# EPICS alarm handler configuration: apps/alhConfig/vacuum.alhConfig
GROUP    NULL                         VACUUM
CHANNEL  VACUUM                       hallb_VCG2C21Tr
$COMMAND  medm -x -attach -cmap -macro "sig=hallb_VCG2C21Tr" aiaocalc_alarm.adl >> /dev/null
$ALARMCOUNTFILTER  99 60
$GUIDANCE
                The cold cathode gauge at the moller region is out of spec.
                This means the vacuum between the shield wall and the tagger
                magnet has degraded.  Use the MYA Viewer and monitor the hallb_VCG2C21Tr
                to check for trends in the past few hours.  If the vacuum is degrading (values increasing on
                the plots) then contact engineering on call.   Also contact MCC and inform them about the
                problem, they might want to shut off the beam and close some valves to isolate the problem.
                If the vacuum spiked and recovered, continue taking
                data.
$END
CHANNEL  VACUUM                       hallb_VCG2C21ATr
$COMMAND  medm -x -attach -cmap -macro "sig=hallb_VCG2C21ATr" aiaocalc_alarm.adl >> /dev/null
$ALARMCOUNTFILTER  99 60
$GUIDANCE
                The cold cathode gauge at the moller region is out of spec.
                This means the vacuum between the shield wall and the tagger
                magnet has degraded.  Use the MYA Viewer and monitor the hallb_VCG2C21ATr
                to check for trends in the past few hours.  If the vacuum is degrading (values increasing on
                the plots) then contact engineering on call.   Also contact MCC and inform them about the
                problem, they might want to shut off the beam and close some valves to isolate the problem.
                If the vacuum spiked and recovered, continue taking
                data.
$END
CHANNEL  VACUUM                       hallb_VCG2C24ATr
$COMMAND  medm -x -attach -cmap -macro "sig=hallb_VCG2C24ATr" aiaocalc_alarm.adl >> /dev/null
$ALARMCOUNTFILTER  99 60
$GUIDANCE
                The tagger turbo speed is below operating range...it may have tripped off.
                Use the MYA Viewer and monitor hallb_VCG2C24ATr
                to check for trends in the past few hours.  If the vacuum is degrading (values increasing on
                the plots) then contact engineering on call.   Also contact MCC and inform them about the
                problem, they might want to shut off the beam and close some valves to isolate the problem.
                If the vacuum spiked and recovered, continue taking
                data.
$END
CHANNEL  VACUUM                       hallb_VCG2H00ATr
$COMMAND  medm -x -attach -cmap -macro "sig=hallb_VCG2H00ATr" aiaocalc_alarm.adl >> /dev/null
$ALARMCOUNTFILTER  99 60
$GUIDANCE
                The cold cathode gauge at 2H00 is out of spec.  This means the vacuum between the tagger magnet
                and target has degraded. Use the MYA Viewer and monitor hallb_VCG2H00ATr
                to check for trends in the past few hours.  If the vacuum is degrading (values increasing on
                the plots) then contact engineering on call.   Also contact MCC and inform them about the
                problem, they might want to shut off the beam and close some valves to isolate the problem.
                If the vacuum spiked and recovered, continue taking
                data.
$END
CHANNEL  VACUUM                       hallb_VCG2H01ATr
$COMMAND  medm -x -attach -cmap -macro "sig=hallb_VCG2H01ATr" aiaocalc_alarm.adl >> /dev/null
$ALARMCOUNTFILTER  99 60
$GUIDANCE
                The cold cathode gauge at 2H01A is out of spec.  This means the vacuum between the tagger
                and target has degraded. Use the MYA Viewer and monitor hallb_VCG2H01ATr
                to check for trends in the past few hours.  If the vacuum is degrading (values increasing on
                the plots) then contact engineering on call.   Also contact MCC and inform them about the
                problem, they might want to shut off the beam and close some valves to isolate the problem.
                If the vacuum spiked and recovered, continue taking
                data.
$END
CHANNEL  VACUUM                       hallb_VCG2H02ATr
$COMMAND  medm -x -attach -cmap -macro "sig=hallb_VCG2H02ATr" aiaocalc_alarm.adl >> /dev/null
$ALARMCOUNTFILTER  99 60
$GUIDANCE
                The cold cathode gauge at 2H02A is out of spec. Use the MYA Viewer and monitor hallb_VCG2H02ATr
                to check for trends in the past few hours.  If the vacuum is degrading (values increasing on
                the plots) then contact engineering on call.   Also contact MCC and inform them about the
                problem, they might want to shut off the beam and close some valves to isolate the problem.
                If the vacuum spiked and recovered, continue taking
                data.
$END
CHANNEL  VACUUM                       HPS_SVT:PLC:i:Vacuum-Value
$COMMAND  medm -x -attach -cmap -macro "sig=HPS_SVT:PLC:i:Vacuum-Value" aiaocalc_alarm.adl >> /dev/null
$ALARMCOUNTFILTER  99 60
$GUIDANCE
                The voltage of the Faraday Cup ION pump is out of spec. Use the MYA Viewer and monitor HPS_SVT:PLC:i:Vacuum-Value
                to check for trends in the past few hours.  If the vacuum is degrading (values increasing on
                the plots) then contact engineering on call.   Also contact MCC and inform them about the
                problem, they might want to shut off the beam and close some valves to isolate the problem.
                If the vacuum spiked and recovered, continue taking
                data.
$END
